FUNCTION_BLOCK FB_WorkerDefGrid_Print EXTENDS FB_WorkerDefGrid
VAR_INPUT
  nEncoderPos           : DINT;   // Absolute virtual encoder
  bHardwareSync         : BOOL;
  bHardwareHold         : BOOL;
  fPrintStartOffset     : LREAL;  //PU->PG/PA offset
  fPrintYOffset         : LREAL;  //Y-Shift in ram memory
  fMasterSpeed          : LREAL;  //Speed [m/s]
  fPUElevation          : LREAL;  //PU distance from substrate [m]
  fPUPlate1_Temperature : LREAL;  // PU Plate1 temperature
  fPUPlate2_Temperature : LREAL;  // PU Plate2 temperature
END_VAR

VAR_OUTPUT
END_VAR

VAR
  _bNewJob           : BOOL;
  sDefGridSettings   : ST_DefGridSettings;  
  fCurrentColumnPos  : LREAL; // Currently column position
  fCurrentPreCharge  : LREAL; // Currently to be precharged
  nChargedColumns    : UDINT; // Already charged columns

  fbDropSpeedComp    : FB_DropSpeedComp;  
  fbPs               : FB_PS_Grid;
  fbPa               : FB_PA;
  fB_PcAdapter       : FB_PC_Adapter;

  _pAdsPu            : POINTER TO ST_ADS_PU;      // PU interface
  _pAdsCam           : POINTER TO ST_ADS_CAMERA;  // camera interface PUC
  _fPrintStartOffset : LREAL;   // internal print start offset (distance Cam -> PG1 + PG Offset + PU offset)
  _fWorkerOffset     : LREAL;   // worker offset from X0 static
  _nPosX0            : DINT;    // X0 for last attached CT (detected postion)
  _nPosXS            : DINT;    // XS for last attached CT (shifted print start position)
  _nPosXDelta        : DINT;    // Shift value X0 -> XS
  _fPosY             : LREAL;   // Y shift for last attached CT
  _nPosDeltaToPrint  : DINT;    // delta pos in [SbuPx] from attach to print
  _bPaStarted        : BOOL;
  _bPaStartRequested : BOOL;
  fBStartTimeout     : TON;
  rTrigSync          : R_TRIG;
  _bForceDefGridOff  : BOOL;    // force deformation grid stream to ph off (send 0)
  
  (*grid correction*)
  _fDxGlobalShift    : LREAL;
  _fDyGlobalShift    : LREAL;
  
  (*grid limit*)
  _fLimitCorrectionX : LREAL;     // correction limit in y (abs) [px]
  _fLimitCorrectionY : LREAL;     // correction limit in y (abs) [px]
    
  (*Messaging*)
  _bMsgInitialized   : BOOL;
  fb_MsgQueue        : FB_MSG_QUEUE;                        (*Message queue*)
  fb_MsgHandler      : FB_MSG_HANDLER;                      (*Message handler*)
  sL_MsgConfig       : ST_MSG_CONFIG;                       (*Message config*)
  fb_Msg             : ARRAY [1..iC_NUM_MSG] OF FB_MESSAGE; (*Messages*)
END_VAR

VAR_STAT
  // PU Deformation/correction for all instance
  fbFineAlignement   : FB_FineAlignement;
END_VAR

VAR PERSISTENT
  _fColumnsToPrecharge : LREAL := nC_COLUMNS_TO_PRECHARGE;
  _fStartShiftOffset   : LREAL := fC_START_SHIFT_OFFSET;
  _fStartShiftFactor   : LREAL := fC_START_SHIFT_FACTOR;
END_VAR

VAR CONSTANT
  iC_NUM_MSG               : UDINT := 5;
  nC_COLUMNS_TO_PRECHARGE  : LREAL := 2.1;
  fC_GRIDPOINT_STREAM_TIME : LREAL := 0.0025;     // time to stream one point [s]
  fC_START_SHIFT_FACTOR    : LREAL := -2.4E-2;
  fC_START_SHIFT_OFFSET    : LREAL := -1.0E-2;
END_VAR

IF _pParamMediator = 0 THEN RETURN; F_Report_Error(ErrType:=EN_REPORT_ERROR_TYPE.Report_Error_0Pointer); END_IF

//TODO Add error/warnings
bError := FALSE;
nError := 0;

fbDropSpeedComp(fMasterSpeed:=fMasterSpeed, fDropTravelDistance:=fPUElevation);

//Start offset update
IF _fPrintStartOffset <> (fPrintStartOffset + _pParamMediator^.fCameraToPrintOffset + _pParamMediator^.fDetectToCamera) THEN //Worker position changed
  IF _pAttachedCt = 0 THEN //Update only without attached container
    _fPrintStartOffset :=fPrintStartOffset + _pParamMediator^.fCameraToPrintOffset + _pParamMediator^.fDetectToCamera;
	END_IF
END_IF

//Worker position update
IF _fWorkerPosition <> (_fPrintStartOffset + (_fStartShiftOffset + _fStartShiftFactor * fMasterSpeed)) THEN //Worker position changed (camera settings change)
  IF _pAttachedCt = 0 THEN //Update only without attached container
    // WorkerPosition =  PU<-CAM + CAM<-SheetDetect + StartShift calculated (with speed)
    fPosition := _fPrintStartOffset + (_fStartShiftOffset + _fStartShiftFactor * fMasterSpeed);
	END_IF
END_IF

(*---- Messaging -----------------------*)
IF _bMsgInitialized THEN
  fb_MsgHandler();
  {warning 'TODO: implement PrintWorker & PG messages'}
  //fB_Msg[1](bI_Status := dfsdfdsf);
  fb_MsgQueue();
END_IF

PROPERTY aPaState : STRING
GET
aPaState := fbPa.aPaState;
END_GET
END_PROPERTY

METHOD PROTECTED  Attach : BOOL
VAR_INPUT
  iCT              : I_CT;                         (*container at triggered event position*)
END_VAR

VAR
  nConvErr        : UDINT;
END_VAR
Attach:=FALSE;

IF SUPER^.Attach(iCT:=iCT) THEN
  // Additional worker checks
    // - job is valid?
  IF _pAttachedCt^.pJob = 0 OR NOT _bJobActive THEN
    Release(iCT:=iCT);
    RETURN;   // do not print
  
  // CT valid & CT present
  ELSIF NOT _pAttachedCt^.bValid OR NOT _pAttachedCt^.bProductPresent THEN
    Release(iCT:=iCT);
    RETURN;   // do not print
  
  // Ignore start due to hardware hold  
  ELSIF bHardwareHold THEN
    _pAttachedCt^.setError(ErrDef:=EC_Print.ecPaAbortHold, Src:=_pEcSrc^);
    Release(iCT:=iCT);
    RETURN;   // do not print
  
  // - OK attach
  ELSE
    Attach := TRUE;
	END_IF
  
  
  //Prepare print station
  fbPs.bPrintEnable := iCT.bValid AND iCT.bProductPresent;
  fbPs.setGrid(sGrid:=sDefGridSettings);
  nChargedColumns := 0;
  _fDxGlobalShift := _pAttachedCt^.fDxShift;
  _fDyGlobalShift := _pAttachedCt^.fDyShift;

  //Start print, PA should be in READY or DONE
  
  // Set X print position
  _nPosX0 :=    _pAttachedCt^.getPosX0(nPosDomain:=E_PosDomain.master_pos)
              //- General Shift
              - F_MeterToSubPixel(fbDropSpeedComp.fDropPlacementError,_fPrintResolution*_fSubPxResolution); // - drop compensation*)
  _nPosXDelta := F_MeterToSubPixel(_fPrintStartOffset,_fPrintResolution*_fSubPxResolution); // + PG/PA Shift (additional PG offset 0 for firstLine)

  IF GVL_Deformation.bC_UseGlobalGridShift THEN
    _nPosXDelta := _nPosXDelta + FC_LREAL_TO_DINT(_fDxGlobalShift, ADR(nConvErr));                  // + global shift from grid points
  END_IF

  _nPosXS := _nPosX0 + _nPosXDelta;
  fB_PcAdapter.setPrintStartPos(nX0:=_nPosXS);
  
  // Set Y print position
  _fPosY := fPrintYOffset;
  IF GVL_Deformation.bC_UseGlobalGridShift THEN
    _fPosY := _fPosY + _fDyGlobalShift;    // + global shift from grid points
  END_IF
  fB_PcAdapter.setPrintYShift(nYShift:=FC_LREAL_TO_DINT(_fPosY, ADR(nConvErr)));

  // check
  IF _nPosXS < nEncoderPos THEN
    LogWarning(Msg:='Print start position < Encoder position');
	END_IF
  
  // save current distance to print position
  _nPosDeltaToPrint := _nPosXS - iCT.GetPos(nPosDomain:=E_PosDomain.master_pos) - _nPosX0;
  checkGridTiming();
  
  IF fbPa.printStart() THEN
    _bPaStarted := FALSE;
    _bPaStartRequested := TRUE;
    Attach:=TRUE;
    LogLvl(Lvl:=E_LogSeverity.Debug, F_Concat2('printStart:', _pAttachedCt^.print(0)));  // print container
    LogLvl(Lvl:=E_LogSeverity.Debug, F_Concat4('> XS:', TO_STRING(_nPosXS), ' = X0:', TO_STRING(_pAttachedCt^.GetPosX0(nPosDomain:=E_PosDomain.master_pos))));
    IF GVL_Deformation.bC_UseGlobalGridShift THEN
      LogLvl(Lvl:=E_LogSeverity.Debug, F_Concat6('> + shDx:', TO_STRING(_fDxGlobalShift), 
                                                 ' + shStartOffs:', TO_STRING(F_MeterToSubPixel(_fPrintStartOffset,_fPrintResolution*_fSubPxResolution)),
                                                 ' - shDropComp:', TO_STRING(F_MeterToSubPixel(fbDropSpeedComp.fDropPlacementError,_fPrintResolution*_fSubPxResolution))
                                                 ));
    ELSE
      LogLvl(Lvl:=E_LogSeverity.Debug, F_Concat4( 
                                           ' + shStartOffs:', TO_STRING(F_MeterToSubPixel(_fPrintStartOffset,_fPrintResolution*_fSubPxResolution)),
                                           ' - shDropComp:', TO_STRING(F_MeterToSubPixel(fbDropSpeedComp.fDropPlacementError,_fPrintResolution*_fSubPxResolution))
                                           ));
		END_IF
  ELSE  
    LogError(Msg:='PA not ready to start at attach');
    Release(iCT := iCT);
	END_IF
  
ELSE
  // parent attach failed case
END_IF
END_METHOD

METHOD PRIVATE checkGridTiming : BOOL
VAR
END_VAR
// check for timing problems
IF fMasterSpeed <> 0 THEN

  // - check pre-charge at beginning
  IF _fColumnsToPrecharge * fC_GRIDPOINT_STREAM_TIME * GVL_Deformation.nC_GridRoiRows >= F_SubPixelToMeter(lPosSubPx:=_nPosDeltaToPrint, fResSubPx:=_fPrintResolution*_fSubPxResolution) / fMasterSpeed  THEN
       LogError('Machine too fast for grid stream (for pre-charge at attach)');
  END_IF
  
 // - check charge time needed per columns vs machine speed and grid-sizeY
 IF GVL_Deformation.nC_GridRoiRows * fC_GRIDPOINT_STREAM_TIME >= F_SubPixelToMeter(lPosSubPx:=TO_DINT(sDefGridSettings.nGridPitchX), fResSubPx:=_fPrintResolution) / fMasterSpeed THEN
   LogError('Machine too fast for grid stream (time rows per column)');
 END_IF

END_IF
END_METHOD

(*
  Limit correction to boundaries
  :return: TRUE if limited
*)
METHOD PRIVATE correctionLimit : BOOL
VAR_INPUT
  pPoint : POINTER TO ST_DeformationPointAccurate;
END_VAR
VAR
  bLimited : BOOL;
  nExeedX, nExeedY : LREAL;
END_VAR
// limit point correction to boundaries and inform
IF    pPoint^.dx >= _fLimitCorrectionX    THEN nExeedX := pPoint^.dx; pPoint^.dx := _fLimitCorrectionX;    bLimited:=TRUE; 
ELSIF pPoint^.dx <= -1*_fLimitCorrectionX THEN nExeedX := pPoint^.dx; pPoint^.dx := -1*_fLimitCorrectionX; bLimited:=TRUE;
ELSIF pPoint^.dy >= _fLimitCorrectionY    THEN nExeedY := pPoint^.dy; pPoint^.dy := _fLimitCorrectionY;    bLimited:=TRUE;
ELSIF pPoint^.dy <= -1*_fLimitCorrectionY THEN nExeedY := pPoint^.dy; pPoint^.dy := -1*_fLimitCorrectionY; bLimited:=TRUE;
END_IF
IF bLimited THEN 
  LogLvl(Lvl:=E_LogSeverity.Warning, Msg:=F_Concat5( 'Point=',TO_STRING(pPoint^.index),
                                                     F_Concat5(' c:r(',TO_STRING(pPoint^.col),'/',TO_STRING(pPoint^.row), ') '),
                                                     F_Concat4('dx:', TO_STRING(nExeedX), ' dy:', TO_STRING(nExeedY)),
                                                     ' correction exceeded limit')); 
END_IF
correctionLimit := bLimited;
END_METHOD

METHOD PRIVATE correctionUpdate : BOOL
VAR_INPUT
  pPoint : POINTER TO ST_DeformationPointAccurate;
END_VAR

// here apply all PU specific corrections
// - mechanical stretch based on temperature extension (if not done in Camera)
// - banana correction
// - Y-shifts of PU
// - trapzedoial correction
// - ...

// global dx/dy correction
//   remove global shift from GridPoints (shifted by PU)
IF GVL_Deformation.bC_UseGlobalGridShift THEN
  pPoint^.dx := pPoint^.dx - _fDxGlobalShift;
  pPoint^.dy := pPoint^.dy - _fDyGlobalShift;
END_IF

// PU Deformation correction
IF GVL_Deformation.bC_UsePUDeformation THEN
  fbFineAlignement.updateCorrection(pPoint:=pPoint);
END_IF
END_METHOD

{attribute 'monitoring':='call'}
PROPERTY fStartShiftFactor : LREAL
GET
fStartShiftFactor := _fStartShiftFactor;
END_GET
SET
_fStartShiftFactor := fStartShiftFactor;
END_SET
END_PROPERTY

{attribute 'monitoring':='call'}
PROPERTY fStartShiftOffset : LREAL
GET
fStartShiftOffset := _fStartShiftOffset;
END_GET
SET
_fStartShiftOffset := fStartShiftOffset;
END_SET
END_PROPERTY

METHOD PROTECTED gridUpdate : BOOL
VAR_INPUT
  bEnableDeformation : BOOL;      // enable correction update, else correction (0/0) is written
END_VAR
VAR
  sPoint : ST_DeformationPointAccurate;
  nRow : UDINT;
  nAvailPoints : UDINT;
  nConvErr : UDINT;
END_VAR
VAR_INST
  nAvailPoints_mem : UDINT;
END_VAR
//TODO: rewrite this method to look cleaner (less if else)
gridUpdate:=TRUE;

// calculate grid column position
IF sDefGridSettings.nGridPitchX <> 0 THEN
  fCurrentColumnPos := fCtPosition / (sDefGridSettings.nGridPitchX * _fSubPxResolution);   // calc grid column position relative to worker
END_IF

//Check for next correction update 
IF fCurrentColumnPos + _fColumnsToPrecharge > nChargedColumns AND nChargedColumns <= sDefGridSettings.nGridSizeX THEN
  IF bEnableDeformation THEN 
    // sync deformation points
    fCurrentPreCharge := fCurrentColumnPos + _fColumnsToPrecharge;
    WHILE FLOOR(fCurrentPreCharge) > nChargedColumns AND nChargedColumns <= sDefGridSettings.nGridSizeX DO
      nAvailPoints := _pAttachedCt^.nAvailableGridPoints;
      IF nAvailPoints >= sDefGridSettings.nGridSizeY * (nChargedColumns+1) THEN // Complete column available?
        nAvailPoints_mem := 0;
        LogLvl(Lvl:=E_LogSeverity.Debug, Msg:=F_Concat2('Charge CG col: ',TO_STRING(nChargedColumns)));
        FOR nRow := 0 TO sDefGridSettings.nGridSizeY - 1 DO
          // get points
          IF _pAttachedCt^.getDeformationPoint(nCol:=nChargedColumns, nRow:=nRow, sPoint => sPoint) THEN
            // transfer the displacement into a correction
            sPoint.dx := sPoint.dx;
            sPoint.dy := sPoint.dy;
            
            // apply PU corrections
            correctionUpdate(pPoint:=ADR(sPoint));
            
            // correction limitation
            correctionLimit(pPoint:=ADR(sPoint));
            
            // send point
            IF NOT fbPs.newGridPoint(sPoint:=sPoint) THEN
               LogError(Msg:='stream new point failed');
               gridUpdate:=FALSE;
               RETURN;
            END_IF
          ELSE
            LogError(Msg:='get new grid point failed');
            gridUpdate:=FALSE;
          END_IF
        END_FOR
        
        nChargedColumns := nChargedColumns + 1;
      ELSE
        IF nAvailPoints > nAvailPoints_mem THEN // log once or after every update of new available poinst
          LogError(Msg:='point column expected but not available');
        END_IF
        nAvailPoints_mem := nAvailPoints;
        gridUpdate:=FALSE;
        RETURN;
      END_IF 
    END_WHILE
  ELSE
    // send points with no deformation
      FOR nRow := 0 TO sDefGridSettings.nGridSizeY - 1 DO
        MEMSET(destAddr:=ADR(sPoint), fillByte:=0, n:=SIZEOF(sPoint));
        sPoint.col := TO_DINT(nChargedColumns);
        sPoint.row := TO_DINT(nRow);
        IF NOT fbPs.newGridPoint(sPoint:=sPoint) THEN
           LogError(Msg:='stream new point failed');
           gridUpdate:=FALSE;
           RETURN;
        END_IF
    END_FOR
    nChargedColumns := nChargedColumns + 1;
	END_IF
END_IF
END_METHOD

METHOD InitAds
VAR_INPUT
  pAdsIfCam  : POINTER TO ST_ADS_CAMERA;
  pAdsIfPu   : POINTER TO ST_ADS_PU;
END_VAR
_pAdsCam := pAdsIfCam;
_pAdsPu  := pAdsIfPu;
END_METHOD

METHOD InitMsg : BOOL
VAR_INPUT
  pMsgInterface : POINTER TO ST_ADS_MSG_IF;
END_VAR
VAR
  nCtr : UDINT;
END_VAR
IF pMsgInterface = 0 THEN RETURN; END_IF

(*Messaging*)
sL_MsgConfig.bI_Enable       := TRUE;
sL_MsgConfig.pI_FbMsgHandler := ADR(fb_MsgHandler);
fb_MsgHandler.pI_MsgQueue    := ADR(fb_MsgQueue);
fb_MsgQueue.pI_MsgInterface  := pMsgInterface;
fb_MsgQueue.cI_MaxElement    := 6;

(*Messages*)
FOR nCtr := 1 TO iC_NUM_MSG DO
  fb_Msg[nCtr].pI_MsgConfig       := ADR(sL_MsgConfig);
  fb_Msg[nCtr].iI_MsgLocation     := 0;
END_FOR
//fb_Msg[1].iI_MsgNumber       := ;
// ...

_bMsgInitialized := TRUE;
END_METHOD

METHOD InitWorkerPrint : BOOL
VAR_INPUT
  fPrintUnitWidth   : LREAL;     // print unit width [m]
  fLimitCorrectionX : LREAL;     // correction limit in y (abs) [px]
  fLimitCorrectionY : LREAL;     // correction limit in y (abs) [px]
END_VAR
IF NOT bInitialized                THEN LogError('Base Worker not initialized! call init() before'); RETURN; END_IF
IF (_pAdsCam = 0) OR (_pAdsPu = 0) THEN LogError('Call InitAds() before, ads interface unknown');    RETURN; END_IF

// worker specific init

//Print Aggregate
_fLimitCorrectionX := ABS(fLimitCorrectionX);
_fLimitCorrectionY := ABS(fLimitCorrectionY);

fbPa.bSyncAfterDone := FALSE;
fbPa.init(iPcAdapter := fB_PcAdapter, iPsInterface := fbPs);

fbFineAlignement.init(pAdsCam := _pAdsCam, fPxReso := _fPrintResolution, fPuWidth := fPrintUnitWidth);
END_METHOD

METHOD   mJobStart
VAR_INPUT
	sJobDef	: CalmarCompPrint.I_JobDefinition;
END_VAR
IF NOT bEnable THEN RETURN; END_IF  // only if enabled

fbPa.jobStart();

_bNewJob := TRUE;
_bJobActive := TRUE;

// set correction ref points
_pAdsCam^.sI_CorrectionPointIndication[1].posx := 0;
_pAdsCam^.sI_CorrectionPointIndication[1].posy := 0;
_pAdsCam^.sI_CorrectionPointIndication[2].posx := DINT_TO_REAL(_pAdsPu^.sI_JobSettings.lI_ImageDepth) / 1000;
_pAdsCam^.sI_CorrectionPointIndication[2].posy := 0;
_pAdsCam^.sI_CorrectionPointIndication[3].posx := 0;
_pAdsCam^.sI_CorrectionPointIndication[3].posy := DINT_TO_REAL(_pAdsPu^.sI_JobSettings.lI_ImageWidth) / 1000;
_pAdsCam^.sI_CorrectionPointIndication[4].posx := DINT_TO_REAL(_pAdsPu^.sI_JobSettings.lI_ImageDepth) / 1000;
_pAdsCam^.sI_CorrectionPointIndication[4].posy := DINT_TO_REAL(_pAdsPu^.sI_JobSettings.lI_ImageWidth) / 1000;
END_METHOD

METHOD  mJobStop
VAR_INPUT
	sStatus	: CalmarCompPrint.I_JobStatus;
END_VAR
fbPa.jobStop();
_bJobActive := FALSE;
END_METHOD

METHOD registerPc : BOOL
VAR_INPUT
  iNewPC : I_PC;
END_VAR
registerPc := fB_PcAdapter.registerPc(iNewPC := iNewPC);
END_METHOD

METHOD registerPh : BOOL
VAR_INPUT
    iPH : I_PH;
    iNewCG : I_Correction_Grid;   // correction grid interface
END_VAR
//Attach head to print station
IF iPH <> 0 THEN
  fbPs.registerCG(iNewPh:=iPH, iNewCG:=iNewCG);
END_IF
END_METHOD

PROPERTY sPcFlags : CalmarCompPrint.ST_PC_FLAGS
GET
sPcFlags := fB_PcAdapter.sPcFlags;
END_GET
END_PROPERTY

PROPERTY sPcState :  CalmarCompPrint.ST_PG_STATUS
GET
VAR
  sJobStatus : ST_JobProgress;
END_VAR
sPcState.bStartPrintCanEx := fBPa.bStartCanEx;
sPcState.bStartPrintExec  := fBPa.bStartExec;
sPcState.bStopPrintCanEx  := fBPa.bStopCanEx;
sPcState.bStopPrintExec   := fBPa.bStopExec;
sPcState.bPausePrintCanEx := FALSE;       // obsolete ???
sPcState.bPausePrintExec  := FALSE;       // obsolete ???
sPcState.bReady           := fB_PcAdapter.bAllReady OR fB_PcAdapter.bAllDone;
sPcState.bError           := fB_PcAdapter.bError;
sPcState.bPrinting        := fB_PcAdapter.bAllPrinting;
sPcState.bLoad            := fB_PcAdapter.bAllPreparing;
sPcState.bArmed           := fB_PcAdapter.bAllPrinting OR fB_PcAdapter.bAllReady OR fB_PcAdapter.bAllDone OR fB_PcAdapter.bAllPreparing;
sPcState.bEnabled         := bEnable;
sPcState.bStartStrb       := fBPa.bStartStrb;
sPcState.bPcEnabled       := fB_PcAdapter.bPcEnable;
sPcState.lProductCount    := 0;            // obsolete ???
sPcState.sJobStatus       := sJobStatus;   // obsolete ???
END_GET
END_PROPERTY

METHOD  work
VAR
  bDeformErr : BOOL;
  nDeformStep : E_DeformationStep;
END_VAR
SUPER^.work();

(*new job attached*)
IF _pParamMediator <> 0 AND _bNewJob THEN
  _bNewJob := FALSE;
  sDefGridSettings := _pParamMediator^.sDeformationGridSetttings;
  // fix some potential errors
  IF sDefGridSettings.nGridPitchX = 0 THEN sDefGridSettings.nGridPitchX :=1024; LogError(F_concat2('grid not configured, set default nGridPitchX=',TO_STRING(sDefGridSettings.nGridPitchX))); END_IF
  IF sDefGridSettings.nGridPitchY = 0 THEN sDefGridSettings.nGridPitchY :=1024; LogError(F_concat2('grid not configured, set default nGridPitchY=',TO_STRING(sDefGridSettings.nGridPitchY))); END_IF
END_IF

(*PU deformation*)
IF GVL_Deformation.bC_UsePUDeformation THEN
  fbFineAlignement.fT_PL1 := fPUPlate1_Temperature;
  fbFineAlignement.fT_PL2 := fPUPlate2_Temperature;
  fbFineAlignement();
END_IF

(*Update virtual encoder on all controller boards*)
fB_PcAdapter.setEncoderPos(nEncoderPos);
fB_PcAdapter();

(*Call print aggregate*)
rTrigSync(CLK:=bHardwareSync); 
IF rTrigSync.Q THEN fbPa.sync(); END_IF   // external sync
fbPa.bHold := bHardwareHold;              // external hw hold
fbPa();

fBStartTimeout(IN := _bPaStartRequested,PT := T#60MS);

IF _pAttachedCt <> 0 AND bEnable THEN // Work only with attached container
  
  // check for generic error
  IF _pAttachedCt^.bValid AND bHardwareHold THEN
    // abort during printing
    _pAttachedCt^.setError(ErrDef:=EC_Print.ecPaAbortHold, Src:=_pEcSrc^);
  END_IF

  // Grid update
  bDeformErr := _pAttachedCt^.getDeformationStatus(eDStep=>nDeformStep);
  IF NOT bDeformErr AND nDeformStep >= E_DeformationStep.gridStarted AND NOT _bForceDefGridOff THEN 
    IF NOT gridUpdate(bEnableDeformation:=TRUE) THEN
      _pAttachedCt^.AbortDeformation(sReason:='deformation point update failed', Src:=_pEcSrc^);
    END_IF
  ELSE
    // not started or error already --> erase deformation points
    gridUpdate(bEnableDeformation:=FALSE);
  END_IF  
  
  // PA control
  IF _bPaStartRequested THEN
    IF fbPa.bPrinting THEN
      _bPaStarted := TRUE;
      _bPaStartRequested := FALSE;
    ELSIF fBStartTimeout.Q THEN //Stop print at timeout to make ready for next container
      _bPaStarted := FALSE;
      _bPaStartRequested := FALSE;
      fbPa.printStop();
      _pAttachedCt^.setError(ErrDef:=EC_Print.ecPaStartErr, Src:=_pEcSrc^);
      Release(_pAttachedCt^);
		END_IF
  ELSIF _bPaStarted THEN
    //Release container when all points have been processed
    IF fbPa.bDone OR fbPa.bStop THEN
      _bPaStarted := FALSE;
      Release(_pAttachedCt^);
    (*ELSIF fbpa.bError THEN
      _pAttachedCt^.setError(ErrDef:=EC_Print.ecPaPrintErr, Ident:=0);
      Release(_pAttachedCt^);*)
    END_IF 
	END_IF
END_IF  

(*Logging config*)
fbPa.LogLevel := LogLevel;
fB_PcAdapter.LogLevel := LogLevel;
END_METHOD

END_FUNCTION_BLOCK

(* stored: Version 1.1.0.1, ProductVersion 3.1.4024.9
   POU FB_WorkerDefGrid_Print: Id {a3c0fca9-0a63-49f3-a9fd-25e7fe09223b}, SpecialFunc None
   Folder I_PrintStatusClient: Id {adecc86c-91cf-457b-8558-66ae01f4fccc}
   Property aPaState: Id {eb46f66a-52cc-4aca-b9e2-7eab452224bc}
   Get Get: Id {bd1c86fe-132b-41d1-bebb-2a87f1fec851}
   Method Attach: Id {0707666f-371d-4dbd-816b-7dc7310c7f8c}
   Method checkGridTiming: Id {3c550058-b5da-4dae-8fa1-4b3726d81082}
   Method correctionLimit: Id {2ed13c64-ceeb-468e-94a8-66f7e71e9337}
   Method correctionUpdate: Id {8bb67264-11f6-4085-9e91-42d7f81ce449}
   Property fStartShiftFactor: Id {5b817e72-fc10-4a5c-bb03-f73451d2d422}
   Get Get: Id {88d78a4b-1f70-4339-a40e-3a1219c24d43}
   Set Set: Id {1c331bfd-5c6b-4a5b-a1c6-18eec6bac750}
   Property fStartShiftOffset: Id {00b341c7-6131-40b9-842f-40f71d2a4e7a}
   Get Get: Id {71ec859f-d269-41e6-8353-3c7e149955bf}
   Set Set: Id {94e97dfb-95c1-4869-b84d-41f1eaa05af4}
   Method gridUpdate: Id {fff173d9-25b9-4de5-9c1e-6a9aa7228ab2}
   Method InitAds: Id {700fac9c-ee52-417d-9b1e-ccb8aad2f589}
   Method InitMsg: Id {dfa2c5d7-d315-4391-826a-3f0a13e8b388}
   Method InitWorkerPrint: Id {9e11bfb6-2c3b-4cf3-ab44-81a61cbfe170}
   Method mJobStart: Id {e6930aa0-f0d8-458e-9de3-18f675c41155}
   Method mJobStop: Id {8177ad7c-6de2-4f33-9116-3de9fb737ab6}
   Method registerPc: Id {3c39032f-7920-436e-9283-1f58258455df}
   Method registerPh: Id {a62d8de9-9fbf-4ff4-bfce-d2ac72d680d3}
   Property sPcFlags: Id {fa3ef9be-bfc1-497c-bb3e-5711955c8dd7}
   Get Get: Id {31b278ad-9123-44bc-826c-af82c44e3e58}
   Property sPcState: Id {f1d03b4e-3371-40d0-92fe-ec59b44e18d0}
   Get Get: Id {1766068c-03e2-40da-beb8-caa32f985382}
   Method work: Id {cfb4a899-7ea9-4389-855e-b56f1970d69a} *)
